(* Logix 5000 project; controller Ex_2_16 Emulate 5570 rev 33.11; software revision 33.00 *)
// Drilling machine with two-hand controls

TASK MainTask (continuous, watchdog 500 ms) : MainProgram

MODULES
   Local : Emulate 5570 (ICP 4, rev 33.11)
END_MODULES

VAR_GLOBAL   (* controller tags *)
   B3 : BOOL;   // Sensor_B3_WP
   B3_Lamp : BOOL;   // B3_Sensor_LED
   M1_B1 : BOOL;   // Stop_Sensor_Up
   M1_B2 : BOOL;   // Stop_Sensor_Down
   M1_Downward : BOOL;   // Motor_Downward_Direction
   M1_K1 : BOOL;   // Up_Sensor
   M1_K2 : BOOL;   // Down_Sensor
   M1_Upward : BOOL;   // Motor_Upward_Direction
   S1 : BOOL;   // Push Button S1
   S2 : BOOL;   // Push Button S2
END_VAR

PROGRAM MainProgram   (* main routine MainRoutine *)

ROUTINE MainRoutine   (* ladder *)
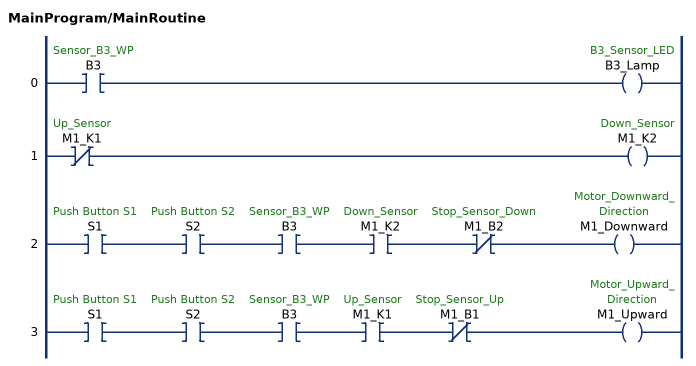
   0: XIC(B3)OTE(B3_Lamp);
   1: XIO(M1_K1)OTE(M1_K2);
   2: XIC(S1)XIC(S2)XIC(B3)XIC(M1_K2)XIO(M1_B2)OTE(M1_Downward);
   3: XIC(S1)XIC(S2)XIC(B3)XIC(M1_K1)XIO(M1_B1)OTE(M1_Upward);
END_ROUTINE
END_PROGRAM
